// TIA Portal V19 export
FUNCTION_BLOCK "A0302_Spintore_FB"   // FB91, LAD
// stored: MemoryReserve 100, SetENOAutomatically false
   VAR_INPUT
      AreaInterface : "AreaInterface";
      ZSI : "udt_ZoneSafetyInterface";
      DSI_Feed : "udt_DeviceSafetyInterface";
      DSI_Valve : "udt_DeviceSafetyInterface";
      Drive : "TAx_DriveInterface";
      DataIn : Struct
         OP : "OP_PB";
         P5 { ExternalAccessible := 'False'; ExternalVisible := 'False'; ExternalWritable := 'False'} : Struct
            Orz_AnalSens : Int;
            FTC_FuoriIngombro_A0301 : Bool;   // FTC fuori ingombro lato bordatrice
         END_STRUCT;
      END_STRUCT;
      Cin : Struct
         Manager { ExternalWritable := 'False'} : Struct
            EnableStopDoorOpeningReq : Bool;
            EnableStopInPhase : Bool;
            EnableStopProgrammed : Bool;
            Control_ON : Bool;
            REST_Req : Bool;
            WORK_Req : Bool;
            Rest : Bool;
            Work : Bool;
         END_STRUCT;
         SemiAut_Pb { ExternalAccessible := 'False'; ExternalVisible := 'False'; ExternalWritable := 'False'} : Bool;
         P4 { ExternalWritable := 'False'} : Struct
            Fermi : "ValveMachine_COut";
         END_STRUCT;
         P5 { ExternalWritable := 'False'} : Struct
            "En/Dis_SpinLat_2" : Bool;   // 1=Enable / 0=Disable
            QuotaIngombro_SpinLat2 : Real;
            QuotaIngombro_SpinLat1 : Real;
            Spintore_Lat : Struct
               Spin_Lat1 : Struct
                  Standstill : Bool;
                  Rest_CheckNext : Bool;
                  Work_CheckNext : Bool;
                  Rest : Bool;
                  Work : Bool;
               END_STRUCT;
               Spin_Lat2 : Struct
                  Standstill : Bool;
                  Rest_CheckNext : Bool;
                  Work_CheckNext : Bool;
                  Rest : Bool;
                  Work : Bool;
               END_STRUCT;
               Vrt_1 : "ValveMachine_COut";
               Orz_1 : "ValveMachine_COut";
               Vrt_2 : "ValveMachine_COut";
               Orz_2 : "ValveMachine_COut";
               Sollevatori : "ValveMachine_COut";
            END_STRUCT;
         END_STRUCT;
         Trasporto { ExternalAccessible := 'False'; ExternalVisible := 'False'; ExternalWritable := 'False'} : "SpeedMachine_COut";
         Bordatrice : Struct   // *************************
            Ax : "Positioning_EPOS_Machine_COut";
            TargetVel : LReal;
            Perc_Vel : LReal;
            Sens : Struct
               FTC_Uscita : Bool;
            END_STRUCT;
         END_STRUCT;
      END_STRUCT;
      Config : Struct
         Ax : "Positioning_EPOS_Machine_Config_NEW";
         Vrt : "ValveMachine_Config";
         Orz : "ValveMachine_Config";
         SpintoreLat : Struct
            QuotaIngombro_SpinLat2 : Real := 2705.0;
            QuotaIngombro_SpinLat1 : Real := 4777.0;
         END_STRUCT;
         Bordatrice : Struct
            QuotaIngresso : Real := 600.0;
         END_STRUCT;
         DelayMissingCondition : Time;
      END_STRUCT;
      HWID_Ax_TEL111 : HW_SUBMODULE;
   END_VAR
   VAR_OUTPUT
      MachineInterface : "MachineInterface";
      DataOut : "Positioning_EPOS_Machine_DataOut";
      COut : Struct
         Ax_Sts : Struct
            PosAttesa_Reached : Bool;
            PosFineSpinta_Reached : Bool;
         END_STRUCT;
         Ax : "Positioning_EPOS_Machine_COut";
         Spintore : "ValveMachine_COut";
         Vrt : "ValveMachine_COut";
         Orz : "ValveMachine_COut";
      END_STRUCT;
   END_VAR
   VAR_IN_OUT
      Par : Struct
         Sens : "Analogic_SensorManagement_Par";
      END_STRUCT;
      Data : Struct
         Sens : "Analogic_SensorManagement_Data";
         HMI : "HMI_Preset";
         Ax_Pos : "A0301_Mach_Ax_Pos_Data";
      END_STRUCT;
      Par_Mach : "A0301_Mach_Sens_Par";
      Par_Ax_Manu : "Positioning_EPOS_Machine_Par";
      Pers_Data : Struct
         EncoderAbsolute_Preset_OK : Bool;
         Persistent_ActualPosition : LReal;
      END_STRUCT;
      Par_Ax_Auto : "A0301_Mach_Speed_Par";
   END_VAR
   VAR
      Alarm : Struct
         Ax : "Positioning_EPOS_Machine_Alr";
         Ax_NeedPreset { S7_SetPoint := 'True'} : Bool;
         Vrt : "ValveAlr";
         Orz : "ValveAlr";
         Orz_AnalSens_Issue : Bool;
         Orz_AnalSens_Compressed : Bool;
      END_STRUCT;
      Warning : Struct
         Ax : "Positioning_EPOS_Machine_Wng";
         Vrt : "ValveMachine_Wng";
         Orz { S7_SetPoint := 'True'} : "ValveMachine_Wng";
         Orz_AnalSens { S7_SetPoint := 'True'} : "Analogic_SensorManagement_Warning";
         OP_REST_MissingCnd : Bool;   // Mancanza comando arresto
         OP_WORK_MissingCnd : Bool;   // Mancanza consenso lavoro
      END_STRUCT;
      Sts : Struct
         ReadyForMove : Bool;   // Pronto al movimento
         OP_CanMoveFreely : Bool;
         OP_Ax_Rest_Cnd : Bool;
         OP_Ax_Work_Cnd : Bool;
         OP_Spin_Rest_Cnd : Bool;
         OP_Spin_Work_Cnd : Bool;
         A0301_Beam_BLean : Real;
         A0302_Beam_BLean : Real;
         Vrt_Work_ExtEnable : Bool;
         Orz_Work_ExtEnable : Bool;
      END_STRUCT;
      Ctrl : Struct
         SpinVrtOrz : Struct
            OP_Rest_Man : Bool;
            OP_Work_Man : Bool;
            OP_Rest_Aut : Bool;
            OP_Work_Aut : Bool;
            OP_Rest : Bool;
            OP_Work : Bool;
         END_STRUCT;
         Ax : Struct
            OP_Rest_Man : Bool;
            OP_Work_Man : Bool;
            OP_Rest_Aut : Bool;
            OP_Work_Aut : Bool;
            OP_Rest : Bool;
            OP_Work : Bool;
            Vel : LReal;
            VelMax : Real;
            Dec : LReal;
         END_STRUCT;
      END_STRUCT;
      HMI : Struct
         Ax : "AnalogSens_HmiData";
         Orz_AnalSens_PB_Preset { ExternalAccessible := 'False'; ExternalVisible := 'False'; ExternalWritable := 'False'} : Bool;   // Pulsante Preset value
         Orz_AnalSens_Preset_Value : LReal;
      END_STRUCT;
      Ax { S7_SetPoint := 'True'} : "Positioning_EPOS_Machine_FB_NEW";   // Spintore longitudinale
      Vrt { S7_SetPoint := 'True'} : "ValveMachine_FB";   // Sollevatore verticale
      Orz { S7_SetPoint := 'True'} : "ValveMachine_FB";   // Compensatore orizzontale
      Orz_AnalSens { S7_SetPoint := 'True'} : "Analogic_SensorManagement";
      ValueBLeanOvr : Array[1..15] of Real;
      IEC : Struct
         TON_DelayFTC_Ingombro_A0301 : IEC_TIMER;
         TOF_DelayFTC_Ingombro_A0301 { S7_SetPoint := 'True'} : IEC_TIMER;
         FTC_On { S7_SetPoint := 'True'} : Bool;
      END_STRUCT;
      AUX : Struct
         OP_Rest_PB : Bool;
         OP_Work_PB : Bool;
      END_STRUCT;
      TON_OP_REST_MissingCnd { S7_SetPoint := 'True'} : TON_TIME;
      TON_OP_WORK_MissingCnd { S7_SetPoint := 'True'} : TON_TIME;
      BTrk_Item : Struct
         BLean : Real;
         O_ID : DInt;
      END_STRUCT;
   END_VAR
   VAR_TEMP
      i : Int;
      DecMax : LReal;
      Orz_SpazioSafe : LReal;
      Calcoli : Struct
         SUB_SpinLat2 : LReal;
         SUB_SpinLat1 : LReal;
         Pos_Target_2 : LReal;
         Pos_Target_1 : LReal;
         Ax_Target : LReal;
      END_STRUCT;
      PE : Struct
         OP_Rest_PB : Bool;
         OP_Work_PB : Bool;
      END_STRUCT;
      BTrk_GetData_A0302 : Struct
         indx : Int;   // Se trovato tra i TODO / ENDING / OUT questo è l'indice dove sono stati prelevati i dati
         Sts : Int;   // 0 = Non Trovato; 0 = ACT; 1 = TODO; 2=ENDING; 3 = OUT
         Item : "Prod_Item_small";
      END_STRUCT;
      BTrk_GetData_A0301 : Struct
         indx : Int;   // Se trovato tra i TODO / ENDING / OUT questo è l'indice dove sono stati prelevati i dati
         Sts : Int;   // 0 = Non Trovato; 0 = ACT; 1 = TODO; 2=ENDING; 3 = OUT
         Item : "Prod_Item_small";
      END_STRUCT;
      Stop_Ax_SpinLong : Bool;
      GetData_A0301_B : Bool;
      GetData_A0302_In : Bool;
   END_VAR
   VAR CONSTANT
      Offset_SpinLong_To_SpinLat2 : Real;   // Offset calcolato da quota ingombro Spintore Laterale2 per bloccare Spintore Longitudinale e allarme se SpinLat2 alto
      Offset_SpinLong_To_SpinLat1 : Real;   // Offset calcolato da quota ingombro Spintore Laterale1 per bloccare Spintore Longitudinale e allarme se SpinLat1 alto
   END_VAR
   // Orz_AnalSens.Filter.Tau := T#10ms;
   VAR_TEMP   // added for the SCL form of the ladder/FBD networks
      _w1 : Bool;
      _w2 : Bool;
      _w3 : Bool;
      _w4 : Bool;
      _w5 : Bool;
      _w6 : Bool;
   END_VAR
BEGIN

REGION Network 1 (SCL): Reset allarmi
   IF #AreaInterface.RstAlarms THEN
       #Alarm.Orz_AnalSens_Issue := FALSE;
       #Warning.Orz_AnalSens.SignalError := FALSE;
   END_IF;
END_REGION

REGION Network 2: <+>
END_REGION

REGION Network 4: CONTROLLO MES lunghezza Beams
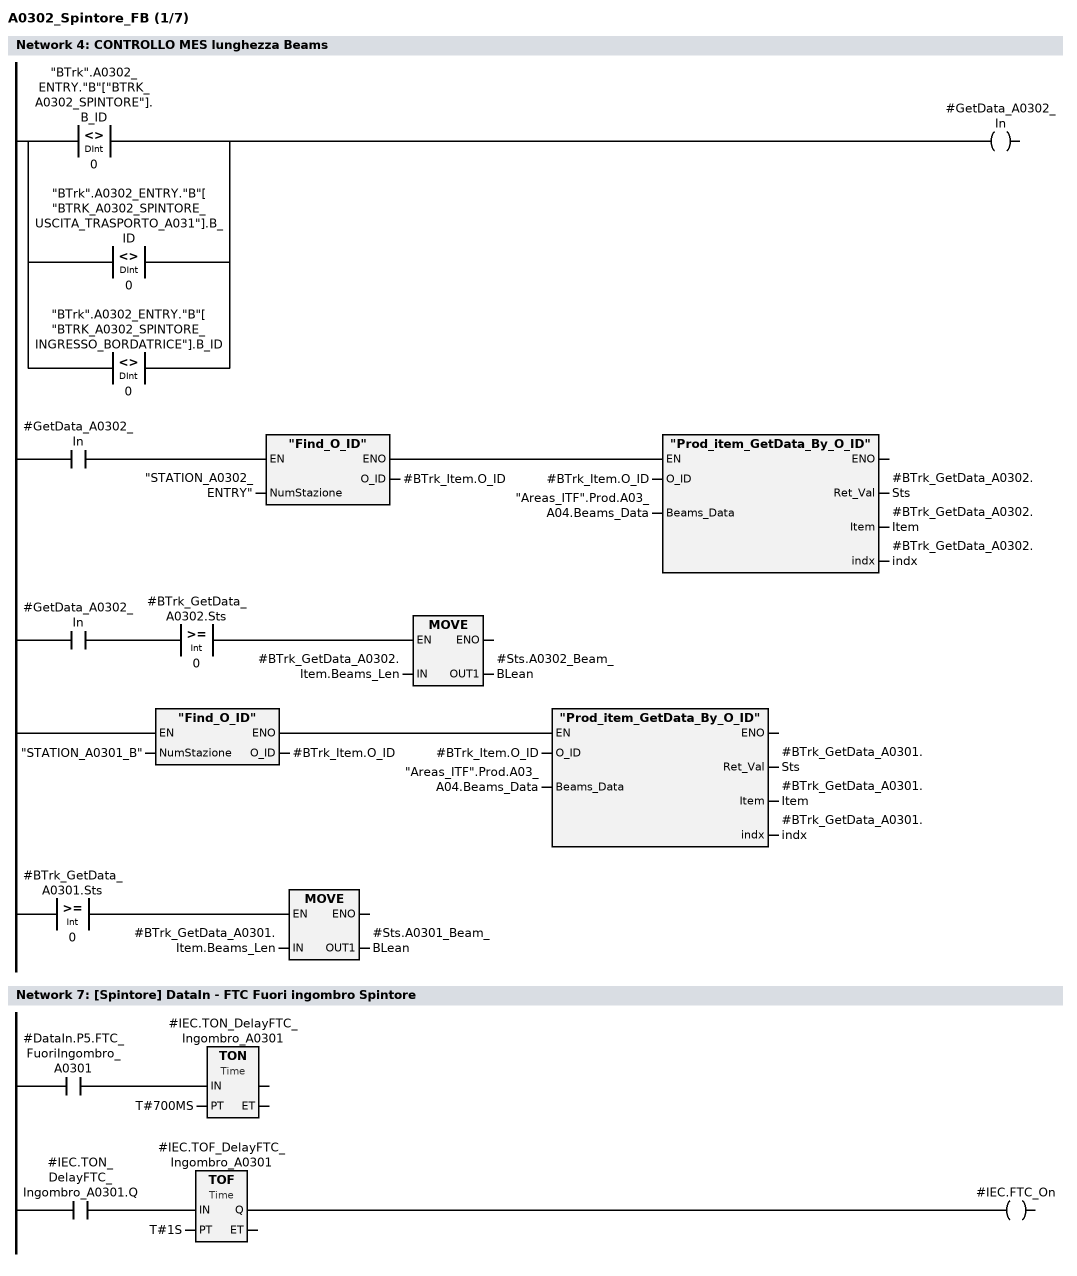
   RUNG wire#powerrail
      { S7_Templates := "SrcType := DInt" } NE_Contact(in1 := "BTrk".A0302_ENTRY."B"["BTRK_A0302_SPINTORE"].B_ID, in2 := 0)
      wire#w1
      Coil( #GetData_A0302_In )
   END_RUNG
   RUNG wire#powerrail
      { S7_Templates := "SrcType := DInt" } NE_Contact(in1 := "BTrk".A0302_ENTRY."B"["BTRK_A0302_SPINTORE_USCITA_TRASPORTO_A031"].B_ID, in2 := 0)
   END_RUNG wire#w1
   RUNG wire#powerrail
      { S7_Templates := "SrcType := DInt" } NE_Contact(in1 := "BTrk".A0302_ENTRY."B"["BTRK_A0302_SPINTORE_INGRESSO_BORDATRICE"].B_ID, in2 := 0)
   END_RUNG wire#w1
   RUNG wire#powerrail
      Contact( #GetData_A0302_In )
      "Find_O_ID"(NumStazione := "STATION_A0302_ENTRY", O_ID => #BTrk_Item.O_ID)
      "Prod_item_GetData_By_O_ID"(O_ID := #BTrk_Item.O_ID, Beams_Data := "Areas_ITF".Prod.A03_A04.Beams_Data, Ret_Val => #BTrk_GetData_A0302.Sts, Item => #BTrk_GetData_A0302.Item, indx => #BTrk_GetData_A0302.indx)
   END_RUNG
   RUNG wire#powerrail
      Contact( #GetData_A0302_In )
      { S7_Templates := "SrcType := Int" } GE_Contact(in1 := #BTrk_GetData_A0302.Sts, in2 := 0)
      Move(in := #BTrk_GetData_A0302.Item.Beams_Len, out1 => #Sts.A0302_Beam_BLean)
   END_RUNG
   RUNG wire#powerrail
      "Find_O_ID"(NumStazione := "STATION_A0301_B", O_ID => #BTrk_Item.O_ID)
      "Prod_item_GetData_By_O_ID"(O_ID := #BTrk_Item.O_ID, Beams_Data := "Areas_ITF".Prod.A03_A04.Beams_Data, Ret_Val => #BTrk_GetData_A0301.Sts, Item => #BTrk_GetData_A0301.Item, indx => #BTrk_GetData_A0301.indx)
   END_RUNG
   RUNG wire#powerrail
      { S7_Templates := "SrcType := Int" } GE_Contact(in1 := #BTrk_GetData_A0301.Sts, in2 := 0)
      Move(in := #BTrk_GetData_A0301.Item.Beams_Len, out1 => #Sts.A0301_Beam_BLean)
   END_RUNG
   // the same network as SCL:
   #GetData_A0302_In := ("BTrk".A0302_ENTRY."B"["BTRK_A0302_SPINTORE"].B_ID <> 0) OR ("BTrk".A0302_ENTRY."B"["BTRK_A0302_SPINTORE_USCITA_TRASPORTO_A031"].B_ID <> 0) OR ("BTrk".A0302_ENTRY."B"["BTRK_A0302_SPINTORE_INGRESSO_BORDATRICE"].B_ID <> 0);
   "Find_O_ID"(EN := #GetData_A0302_In,
               NumStazione := "STATION_A0302_ENTRY",
               O_ID => #BTrk_Item.O_ID,
               ENO => #_w1);
   IF #_w1 THEN
       #BTrk_GetData_A0302.Sts := "Prod_item_GetData_By_O_ID"(O_ID := #BTrk_Item.O_ID,
                               Beams_Data := "Areas_ITF".Prod.A03_A04.Beams_Data,
                               Item => #BTrk_GetData_A0302.Item,
                               indx => #BTrk_GetData_A0302.indx);
   END_IF;
   IF #GetData_A0302_In AND (#BTrk_GetData_A0302.Sts >= 0) THEN
       #Sts.A0302_Beam_BLean := #BTrk_GetData_A0302.Item.Beams_Len;
   END_IF;
   "Find_O_ID"(NumStazione := "STATION_A0301_B", O_ID => #BTrk_Item.O_ID, ENO => #_w2);
   IF #_w2 THEN
       #BTrk_GetData_A0301.Sts := "Prod_item_GetData_By_O_ID"(O_ID := #BTrk_Item.O_ID,
                               Beams_Data := "Areas_ITF".Prod.A03_A04.Beams_Data,
                               Item => #BTrk_GetData_A0301.Item,
                               indx => #BTrk_GetData_A0301.indx);
   END_IF;
   IF #BTrk_GetData_A0301.Sts >= 0 THEN #Sts.A0301_Beam_BLean := #BTrk_GetData_A0301.Item.Beams_Len; END_IF;
END_REGION

REGION Network 5 (SCL): CALCOLI - Posizioni Attesa / Spinta per lavoro Spintore

   #BTrk_GetData_A0302.Item.O_ID := #BTrk_GetData_A0302.Item.O_ID;
   #BTrk_Item.BLean:=#BTrk_GetData_A0302.Item.Beams_Len;
   // ***********************************************************************************************************
   // 
   REGION POSIZIONE ATTESA PEZZO IN ENTRATA

       // Se ho una misura traking vado in posizionamento calcolando la misura del Beams più alta + Offset sennò vado indietro fino a pos. minima
       IF #Sts.A0301_Beam_BLean <> 0 THEN
           #Data.Ax_Pos.PosAttesa := (#Ax.COut.MaxPosition -#Sts.A0301_Beam_BLean) - (#Data.Ax_Pos.OffsetPosAttesa - #Config.Bordatrice.QuotaIngresso);
       ELSIF #Sts.OP_CanMoveFreely THEN
           #BTrk_Item.BLean := 0;
           #Data.Ax_Pos.PosAttesa := ( #Ax.COut.MinPosition) + #Data.Ax_Pos.OffsetPosAttesa;
       END_IF;

   END_REGION ;
   //
   // ***********************************************************************************************************
   // 
   REGION POSIZIONE FINE SPINTA PEZZO IN USCITA

       // CALCOLO Pos.Fine Spinta Target finale
       IF #Sts.A0302_Beam_BLean <> 0 THEN
           #Data.Ax_Pos.PosFineSpinta := (#Ax.COut.MaxPosition - #Sts.A0302_Beam_BLean) + (#Config.Bordatrice.QuotaIngresso);
       ELSIF #BTrk_Item.BLean = 0 THEN
           #Data.Ax_Pos.PosFineSpinta := (#Ax.COut.MaxPosition - #Data.Ax_Pos.OffsetPosAttesa);
       END_IF;

       (*
       // CALCOLO differenza tra Pos.Attesa e Quota ingombro Spintore laterale 2 SE incluso 
       IF #Cin.P5."En/Dis_SpinLat_2"
           AND #Ax.COut.ActualPosition < (#Config.SpintoreLat.QuotaIngombro_SpinLat2 +  #Config.SpintoreLat.OffsetPosAttesa) THEN
           #Calcoli.SUB_SpinLat2 :=((#Data.Ax_Pos.PosAttesa) + (#Config.SpintoreLat.QuotaIngombro_SpinLat2));
       END_IF;

       // CALCOLO differenza tra Pos.Attesa e Quota ingombro Spintore laterale 1 
       IF #Ax.COut.ActualPosition > #Config.SpintoreLat.QuotaIngombro_SpinLat1 THEN
           #Calcoli.SUB_SpinLat1 :=((#Data.Ax_Pos.PosAttesa) + (#Config.SpintoreLat.QuotaIngombro_SpinLat1));
       END_IF;

       // CALCOLI Posizioni Target SPINTORI LATERALI
       #Calcoli.Pos_Target_2 := (#Data.Ax_Pos.PosAttesa) + (#Calcoli.SUB_SpinLat2);
       #Calcoli.Pos_Target_1 := (#Data.Ax_Pos.PosAttesa) + (#Calcoli.SUB_SpinLat1);

       // SPINTORE LATERALE 1&2 - AX - POS. Target
       IF #Cin.P5."En/Dis_SpinLat_2"
           AND #Data.Ax_Pos.PosFineSpinta >= #Calcoli.Pos_Target_2 THEN
           #Calcoli.Ax_Target := #Calcoli.Pos_Target_2;
       ELSIF #Data.Ax_Pos.PosFineSpinta >= #Calcoli.Pos_Target_1
           AND #Ax.COut.ActualPosition < (-#Config.SpintoreLat.QuotaIngombro_SpinLat2) THEN
           #Calcoli.Ax_Target := #Calcoli.Pos_Target_1;
       ELSIF #Ax.#COut.ActualPosition < (-#Config.SpintoreLat.QuotaIngombro_SpinLat1) THEN
           #Calcoli.Ax_Target := #Data.Ax_Pos.PosFineSpinta;
       END_IF;
       *)

   END_REGION ;
   //
   // ***********************************************************************************************************
END_REGION

REGION Network 6: <+>
END_REGION

REGION Network 7: [Spintore] DataIn - FTC Fuori ingombro Spintore
   RUNG wire#powerrail
      Contact( #DataIn.P5.FTC_FuoriIngombro_A0301 )
      { S7_Templates := "time_type := Time" } #IEC.TON_DelayFTC_Ingombro_A0301.TON(pt := T#700MS, et =>)
   END_RUNG
   RUNG wire#powerrail
      Contact( #IEC.TON_DelayFTC_Ingombro_A0301.Q )
      { S7_Templates := "time_type := Time" } #IEC.TOF_DelayFTC_Ingombro_A0301.TOF(pt := T#1S, et =>)
      Coil( #IEC.FTC_On )
   END_RUNG
   // the same network as SCL:
   #IEC.TON_DelayFTC_Ingombro_A0301.TON(IN := #DataIn.P5.FTC_FuoriIngombro_A0301, PT := T#700MS);
   #IEC.TOF_DelayFTC_Ingombro_A0301.TOF(IN := #IEC.TON_DelayFTC_Ingombro_A0301.Q, PT := T#1S);
   #IEC.FTC_On := #IEC.TOF_DelayFTC_Ingombro_A0301.Q;
END_REGION

REGION Network 8: <+>
END_REGION

REGION Network 9: Operazione può muoversi liberamente perchè non sposta nessun BEAM
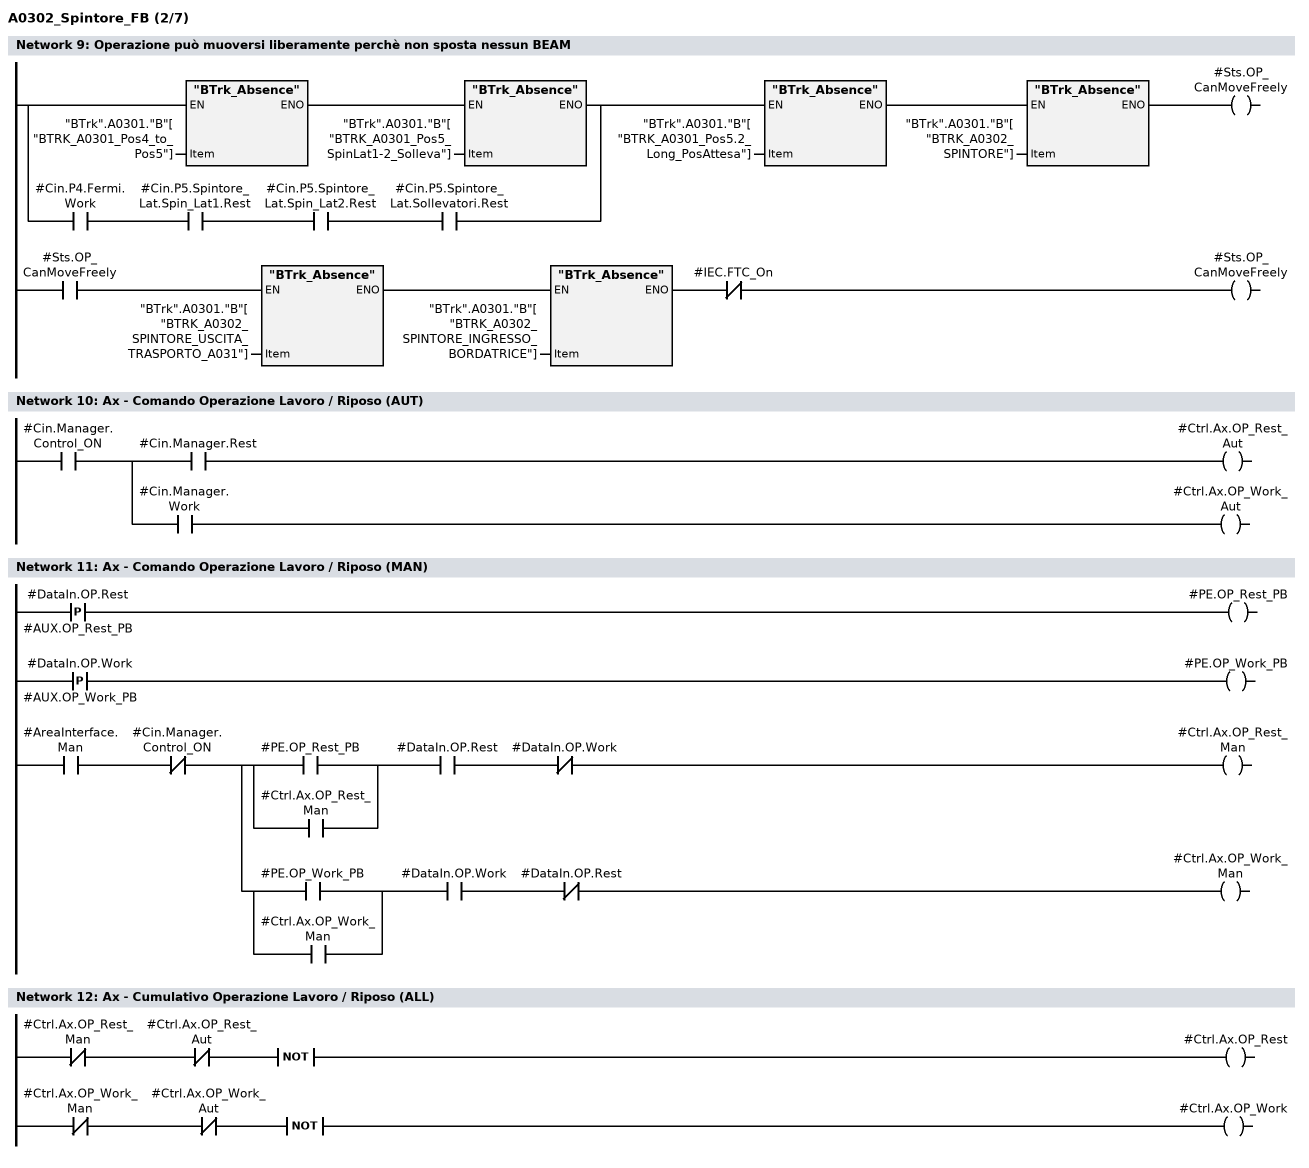
   RUNG wire#powerrail
      "BTrk_Absence"(Item := "BTrk".A0301."B"["BTRK_A0301_Pos4_to_Pos5"])
      "BTrk_Absence"(Item := "BTrk".A0301."B"["BTRK_A0301_Pos5_SpinLat1-2_Solleva"])
      wire#w1
      "BTrk_Absence"(Item := "BTrk".A0301."B"["BTRK_A0301_Pos5.2_Long_PosAttesa"])
      "BTrk_Absence"(Item := "BTrk".A0301."B"["BTRK_A0302_SPINTORE"])
      Coil( #Sts.OP_CanMoveFreely )
   END_RUNG
   RUNG wire#powerrail
      Contact( #Cin.P4.Fermi.Work )
      Contact( #Cin.P5.Spintore_Lat.Spin_Lat1.Rest )
      Contact( #Cin.P5.Spintore_Lat.Spin_Lat2.Rest )
      Contact( #Cin.P5.Spintore_Lat.Sollevatori.Rest )
   END_RUNG wire#w1
   RUNG wire#powerrail
      Contact( #Sts.OP_CanMoveFreely )
      "BTrk_Absence"(Item := "BTrk".A0301."B"["BTRK_A0302_SPINTORE_USCITA_TRASPORTO_A031"])
      "BTrk_Absence"(Item := "BTrk".A0301."B"["BTRK_A0302_SPINTORE_INGRESSO_BORDATRICE"])
      I_Contact( #IEC.FTC_On )
      Coil( #Sts.OP_CanMoveFreely )
   END_RUNG
   // the same network as SCL:
   "BTrk_Absence"(Item := "BTrk".A0301."B"["BTRK_A0301_Pos4_to_Pos5"], ENO => #_w1);
   "BTrk_Absence"(EN := #_w1, Item := "BTrk".A0301."B"["BTRK_A0301_Pos5_SpinLat1-2_Solleva"], ENO => #_w2);
   "BTrk_Absence"(EN := #_w2 OR (#Cin.P4.Fermi.Work AND #Cin.P5.Spintore_Lat.Spin_Lat1.Rest AND #Cin.P5.Spintore_Lat.Spin_Lat2.Rest AND #Cin.P5.Spintore_Lat.Sollevatori.Rest),
                  Item := "BTrk".A0301."B"["BTRK_A0301_Pos5.2_Long_PosAttesa"],
                  ENO => #_w3);
   "BTrk_Absence"(EN := #_w3, Item := "BTrk".A0301."B"["BTRK_A0302_SPINTORE"], ENO => #_w4);
   #Sts.OP_CanMoveFreely := #_w4;
   "BTrk_Absence"(EN := #Sts.OP_CanMoveFreely,
                  Item := "BTrk".A0301."B"["BTRK_A0302_SPINTORE_USCITA_TRASPORTO_A031"],
                  ENO => #_w5);
   "BTrk_Absence"(EN := #_w5, Item := "BTrk".A0301."B"["BTRK_A0302_SPINTORE_INGRESSO_BORDATRICE"], ENO => #_w6);
   #Sts.OP_CanMoveFreely := #_w6 AND NOT #IEC.FTC_On;
END_REGION

REGION Network 10: Ax - Comando Operazione Lavoro / Riposo (AUT)
   RUNG wire#powerrail
      Contact( #Cin.Manager.Control_ON )
      wire#w1
      Contact( #Cin.Manager.Rest )
      Coil( #Ctrl.Ax.OP_Rest_Aut )
   END_RUNG
   RUNG wire#w1
      Contact( #Cin.Manager.Work )
      Coil( #Ctrl.Ax.OP_Work_Aut )
   END_RUNG
   // the same network as SCL:
   #Ctrl.Ax.OP_Rest_Aut := #Cin.Manager.Control_ON AND #Cin.Manager.Rest;
   #Ctrl.Ax.OP_Work_Aut := #Cin.Manager.Control_ON AND #Cin.Manager.Work;
END_REGION

REGION Network 11: Ax - Comando Operazione Lavoro / Riposo (MAN)
   RUNG wire#powerrail
      P_Contact(operand := #DataIn.OP.Rest, bit := #AUX.OP_Rest_PB)
      Coil( #PE.OP_Rest_PB )
   END_RUNG
   RUNG wire#powerrail
      P_Contact(operand := #DataIn.OP.Work, bit := #AUX.OP_Work_PB)
      Coil( #PE.OP_Work_PB )
   END_RUNG
   RUNG wire#powerrail
      Contact( #AreaInterface.Man )
      I_Contact( #Cin.Manager.Control_ON )
      wire#w1
      Contact( #PE.OP_Rest_PB )
      wire#w2
      Contact( #DataIn.OP.Rest )
      I_Contact( #DataIn.OP.Work )
      Coil( #Ctrl.Ax.OP_Rest_Man )
   END_RUNG
   RUNG wire#w1
      Contact( #Ctrl.Ax.OP_Rest_Man )
   END_RUNG wire#w2
   RUNG wire#w1
      Contact( #PE.OP_Work_PB )
      wire#w3
      Contact( #DataIn.OP.Work )
      I_Contact( #DataIn.OP.Rest )
      Coil( #Ctrl.Ax.OP_Work_Man )
   END_RUNG
   RUNG wire#w1
      Contact( #Ctrl.Ax.OP_Work_Man )
   END_RUNG wire#w3
   // the same network as SCL:
   #_w1 := #DataIn.OP.Rest AND NOT #AUX.OP_Rest_PB;   // rising edge of #DataIn.OP.Rest
   #AUX.OP_Rest_PB := #DataIn.OP.Rest;
   #PE.OP_Rest_PB := #_w1;
   #_w2 := #DataIn.OP.Work AND NOT #AUX.OP_Work_PB;   // rising edge of #DataIn.OP.Work
   #AUX.OP_Work_PB := #DataIn.OP.Work;
   #PE.OP_Work_PB := #_w2;
   #_w3 := #AreaInterface.Man AND NOT #Cin.Manager.Control_ON;
   #Ctrl.Ax.OP_Rest_Man := #_w3 AND (#PE.OP_Rest_PB OR #Ctrl.Ax.OP_Rest_Man) AND #DataIn.OP.Rest AND NOT #DataIn.OP.Work;
   #Ctrl.Ax.OP_Work_Man := #_w3 AND (#PE.OP_Work_PB OR #Ctrl.Ax.OP_Work_Man) AND #DataIn.OP.Work AND NOT #DataIn.OP.Rest;
END_REGION

REGION Network 12: Ax - Cumulativo Operazione Lavoro / Riposo (ALL)
   RUNG wire#powerrail
      I_Contact( #Ctrl.Ax.OP_Rest_Man )
      I_Contact( #Ctrl.Ax.OP_Rest_Aut )
      Not()
      Coil( #Ctrl.Ax.OP_Rest )
   END_RUNG
   RUNG wire#powerrail
      I_Contact( #Ctrl.Ax.OP_Work_Man )
      I_Contact( #Ctrl.Ax.OP_Work_Aut )
      Not()
      Coil( #Ctrl.Ax.OP_Work )
   END_RUNG
   // the same network as SCL:
   #Ctrl.Ax.OP_Rest := NOT (NOT #Ctrl.Ax.OP_Rest_Man AND NOT #Ctrl.Ax.OP_Rest_Aut);
   #Ctrl.Ax.OP_Work := NOT (NOT #Ctrl.Ax.OP_Work_Man AND NOT #Ctrl.Ax.OP_Work_Aut);
END_REGION

REGION Network 13: Ax - Condizioni movimento Operazione a Lavoro / Riposo
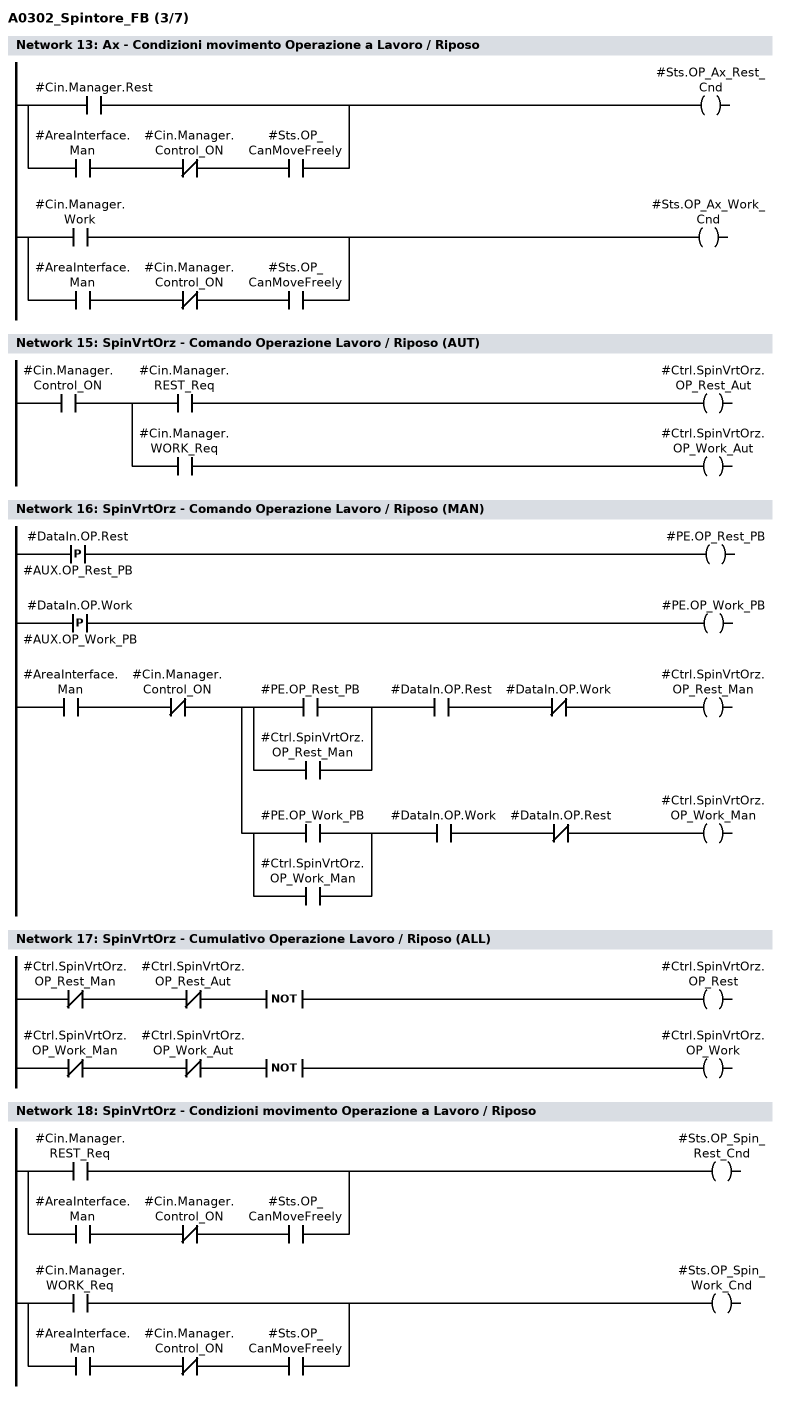
   RUNG wire#powerrail
      Contact( #Cin.Manager.Rest )
      wire#w1
      Coil( #Sts.OP_Ax_Rest_Cnd )
   END_RUNG
   RUNG wire#powerrail
      Contact( #AreaInterface.Man )
      I_Contact( #Cin.Manager.Control_ON )
      Contact( #Sts.OP_CanMoveFreely )
   END_RUNG wire#w1
   RUNG wire#powerrail
      Contact( #Cin.Manager.Work )
      wire#w2
      Coil( #Sts.OP_Ax_Work_Cnd )
   END_RUNG
   RUNG wire#powerrail
      Contact( #AreaInterface.Man )
      I_Contact( #Cin.Manager.Control_ON )
      Contact( #Sts.OP_CanMoveFreely )
   END_RUNG wire#w2
   // the same network as SCL:
   #Sts.OP_Ax_Rest_Cnd := #Cin.Manager.Rest OR (#AreaInterface.Man AND NOT #Cin.Manager.Control_ON AND #Sts.OP_CanMoveFreely);
   #Sts.OP_Ax_Work_Cnd := #Cin.Manager.Work OR (#AreaInterface.Man AND NOT #Cin.Manager.Control_ON AND #Sts.OP_CanMoveFreely);
END_REGION

REGION Network 15: SpinVrtOrz - Comando Operazione Lavoro / Riposo (AUT)
   RUNG wire#powerrail
      Contact( #Cin.Manager.Control_ON )
      wire#w1
      Contact( #Cin.Manager.REST_Req )
      Coil( #Ctrl.SpinVrtOrz.OP_Rest_Aut )
   END_RUNG
   RUNG wire#w1
      Contact( #Cin.Manager.WORK_Req )
      Coil( #Ctrl.SpinVrtOrz.OP_Work_Aut )
   END_RUNG
   // the same network as SCL:
   #Ctrl.SpinVrtOrz.OP_Rest_Aut := #Cin.Manager.Control_ON AND #Cin.Manager.REST_Req;
   #Ctrl.SpinVrtOrz.OP_Work_Aut := #Cin.Manager.Control_ON AND #Cin.Manager.WORK_Req;
END_REGION

REGION Network 16: SpinVrtOrz - Comando Operazione Lavoro / Riposo (MAN)
   RUNG wire#powerrail
      P_Contact(operand := #DataIn.OP.Rest, bit := #AUX.OP_Rest_PB)
      Coil( #PE.OP_Rest_PB )
   END_RUNG
   RUNG wire#powerrail
      P_Contact(operand := #DataIn.OP.Work, bit := #AUX.OP_Work_PB)
      Coil( #PE.OP_Work_PB )
   END_RUNG
   RUNG wire#powerrail
      Contact( #AreaInterface.Man )
      I_Contact( #Cin.Manager.Control_ON )
      wire#w1
      Contact( #PE.OP_Rest_PB )
      wire#w2
      Contact( #DataIn.OP.Rest )
      I_Contact( #DataIn.OP.Work )
      Coil( #Ctrl.SpinVrtOrz.OP_Rest_Man )
   END_RUNG
   RUNG wire#w1
      Contact( #Ctrl.SpinVrtOrz.OP_Rest_Man )
   END_RUNG wire#w2
   RUNG wire#w1
      Contact( #PE.OP_Work_PB )
      wire#w3
      Contact( #DataIn.OP.Work )
      I_Contact( #DataIn.OP.Rest )
      Coil( #Ctrl.SpinVrtOrz.OP_Work_Man )
   END_RUNG
   RUNG wire#w1
      Contact( #Ctrl.SpinVrtOrz.OP_Work_Man )
   END_RUNG wire#w3
   // the same network as SCL:
   #_w1 := #DataIn.OP.Rest AND NOT #AUX.OP_Rest_PB;   // rising edge of #DataIn.OP.Rest
   #AUX.OP_Rest_PB := #DataIn.OP.Rest;
   #PE.OP_Rest_PB := #_w1;
   #_w2 := #DataIn.OP.Work AND NOT #AUX.OP_Work_PB;   // rising edge of #DataIn.OP.Work
   #AUX.OP_Work_PB := #DataIn.OP.Work;
   #PE.OP_Work_PB := #_w2;
   #_w3 := #AreaInterface.Man AND NOT #Cin.Manager.Control_ON;
   #Ctrl.SpinVrtOrz.OP_Rest_Man := #_w3 AND (#PE.OP_Rest_PB OR #Ctrl.SpinVrtOrz.OP_Rest_Man) AND #DataIn.OP.Rest AND NOT #DataIn.OP.Work;
   #Ctrl.SpinVrtOrz.OP_Work_Man := #_w3 AND (#PE.OP_Work_PB OR #Ctrl.SpinVrtOrz.OP_Work_Man) AND #DataIn.OP.Work AND NOT #DataIn.OP.Rest;
END_REGION

REGION Network 17: SpinVrtOrz - Cumulativo Operazione Lavoro / Riposo (ALL)
   RUNG wire#powerrail
      I_Contact( #Ctrl.SpinVrtOrz.OP_Rest_Man )
      I_Contact( #Ctrl.SpinVrtOrz.OP_Rest_Aut )
      Not()
      Coil( #Ctrl.SpinVrtOrz.OP_Rest )
   END_RUNG
   RUNG wire#powerrail
      I_Contact( #Ctrl.SpinVrtOrz.OP_Work_Man )
      I_Contact( #Ctrl.SpinVrtOrz.OP_Work_Aut )
      Not()
      Coil( #Ctrl.SpinVrtOrz.OP_Work )
   END_RUNG
   // the same network as SCL:
   #Ctrl.SpinVrtOrz.OP_Rest := NOT (NOT #Ctrl.SpinVrtOrz.OP_Rest_Man AND NOT #Ctrl.SpinVrtOrz.OP_Rest_Aut);
   #Ctrl.SpinVrtOrz.OP_Work := NOT (NOT #Ctrl.SpinVrtOrz.OP_Work_Man AND NOT #Ctrl.SpinVrtOrz.OP_Work_Aut);
END_REGION

REGION Network 18: SpinVrtOrz - Condizioni movimento Operazione a Lavoro / Riposo
   RUNG wire#powerrail
      Contact( #Cin.Manager.REST_Req )
      wire#w1
      Coil( #Sts.OP_Spin_Rest_Cnd )
   END_RUNG
   RUNG wire#powerrail
      Contact( #AreaInterface.Man )
      I_Contact( #Cin.Manager.Control_ON )
      Contact( #Sts.OP_CanMoveFreely )
   END_RUNG wire#w1
   RUNG wire#powerrail
      Contact( #Cin.Manager.WORK_Req )
      wire#w2
      Coil( #Sts.OP_Spin_Work_Cnd )
   END_RUNG
   RUNG wire#powerrail
      Contact( #AreaInterface.Man )
      I_Contact( #Cin.Manager.Control_ON )
      Contact( #Sts.OP_CanMoveFreely )
   END_RUNG wire#w2
   // the same network as SCL:
   #Sts.OP_Spin_Rest_Cnd := #Cin.Manager.REST_Req OR (#AreaInterface.Man AND NOT #Cin.Manager.Control_ON AND #Sts.OP_CanMoveFreely);
   #Sts.OP_Spin_Work_Cnd := #Cin.Manager.WORK_Req OR (#AreaInterface.Man AND NOT #Cin.Manager.Control_ON AND #Sts.OP_CanMoveFreely);
END_REGION

REGION Network 20 (SCL): Verticale + Orizzontale + Ax - Cin Manager (Esecuzione sequenza comandi)
   #Ax.CIn.Manager.Control_ON:= #Cin.Manager.Control_ON;
   #Orz.Cin.Manager.Control_ON := #Vrt.Cin.Manager.Control_ON := #Cin.Manager.Control_ON;


   #Vrt.Cin.Manager.Rest := FALSE;
   #Vrt.Cin.Manager.Work := FALSE;
   #Orz.Cin.Manager.Rest := FALSE;
   #Orz.Cin.Manager.Work := FALSE;
   #Ax.CIn.Manager.MoveToPos := FALSE;


   // Operazione riposo del cilindro verticale ed orizzontale sullo spintore
   IF (#Ctrl.SpinVrtOrz.OP_Rest OR #Cin.Manager.REST_Req) AND #Sts.OP_Spin_Rest_Cnd THEN

       #Orz.Cin.Manager.Rest := #Orz.COut.Rest := TRUE;
       #Vrt.Cin.Manager.Rest := #Vrt.COut.Rest := #Orz.COut.Rest;

       // Operazione lavoro del cilindro verticale ed orizzontale sullo spintore   
   ELSIF (#Ctrl.SpinVrtOrz.OP_Work OR #Cin.Manager.WORK_Req) AND #Sts.OP_Spin_Work_Cnd THEN

       #Vrt.Cin.Manager.Work := #Vrt.COut.Work := TRUE;
       #Orz.Cin.Manager.Work := #Vrt.Cin.Manager.Work;

   END_IF;

   // Operazione arresto dell' asse spintore quando i 2 ciclindri sono in riposo
   IF #Ctrl.Ax.OP_Rest AND #Sts.OP_Ax_Rest_Cnd THEN
       #Ax.CIn.Manager.Pos := #Data.Ax_Pos.PosAttesa;
       #Ax.CIn.Manager.Vel := #Par_Ax_Auto.Aut_Vel;
       #Ax.CIn.Manager.Acc := #Par_Ax_Auto.Aut_Acc;
       #Ax.CIn.Manager.Dec := #Par_Ax_Auto.Aut_Dec;
       #Ax.CIn.Manager.MoveToPos := TRUE;

       // Se raggiungo la pos.attesa spengo il comando
   ELSIF #Ctrl.Ax.OP_Rest AND #Sts.OP_Ax_Rest_Cnd AND #COut.Ax_Sts.PosAttesa_Reached THEN
       #Ax.CIn.Manager.MoveToPos := #Ax.CIn.Manager.Control_ON := FALSE;

   END_IF;

   // Operazione lavoro dell' asse spintore quando i 2 ciclindri sono in lavoro
   IF #Ctrl.Ax.OP_Work AND #Sts.OP_Ax_Work_Cnd AND #Vrt.COut.Work AND #Orz.COut.Work
        AND NOT #Alarm.Orz_AnalSens_Compressed THEN
       #Ax.CIn.Manager.Pos := #Data.Ax_Pos.PosFineSpinta;
       #Ax.CIn.Manager.Vel := #Par_Ax_Auto.Aut_Vel;
       #Ax.CIn.Manager.Acc := #Par_Ax_Auto.Aut_Acc;
       #Ax.CIn.Manager.Dec := #Par_Ax_Auto.Aut_Dec;
       #Ax.CIn.Manager.MoveToPos := TRUE;

      // Se raggiungo la pos. o il sensore viene compresso disabilito la spinta 
   ELSIF (#Ctrl.Ax.OP_Work AND #Sts.OP_Ax_Work_Cnd) AND #COut.Ax_Sts.PosFineSpinta_Reached THEN
       #Ax.CIn.Manager.MoveToPos := FALSE;

   ELSIF (#Ctrl.Ax.OP_Work AND #Sts.OP_Ax_Work_Cnd) AND #Alarm.Orz_AnalSens_Compressed THEN
       #Ax.CIn.Manager.MoveToPos := FALSE;

   END_IF;
END_REGION

REGION Network 21 (SCL): Verticale + Orizzontale + Ax - CIn Abilitazioni Stop Manager
   #Vrt.Cin.Manager.EnableStopDoorOpeningReq := #Orz.Cin.Manager.EnableStopDoorOpeningReq
   := #Ax.CIn.Manager.EnableStopDoorOpeningReq := #Cin.Manager.EnableStopDoorOpeningReq;

   #Vrt.Cin.Manager.EnableStopInPhase := #Orz.Cin.Manager.EnableStopInPhase
   := #Ax.CIn.Manager.EnableStopInPhase := #Cin.Manager.EnableStopInPhase;

   #Vrt.Cin.Manager.EnableStopProgrammed := #Orz.Cin.Manager.EnableStopProgrammed
   := #Ax.CIn.Manager.EnableStopProgrammed := #Cin.Manager.EnableStopProgrammed;
END_REGION

REGION Network 22: <+>
END_REGION

REGION Network 23: Warning manacanza condizioni esecuzione Operazione RIPOSO / LAVORO
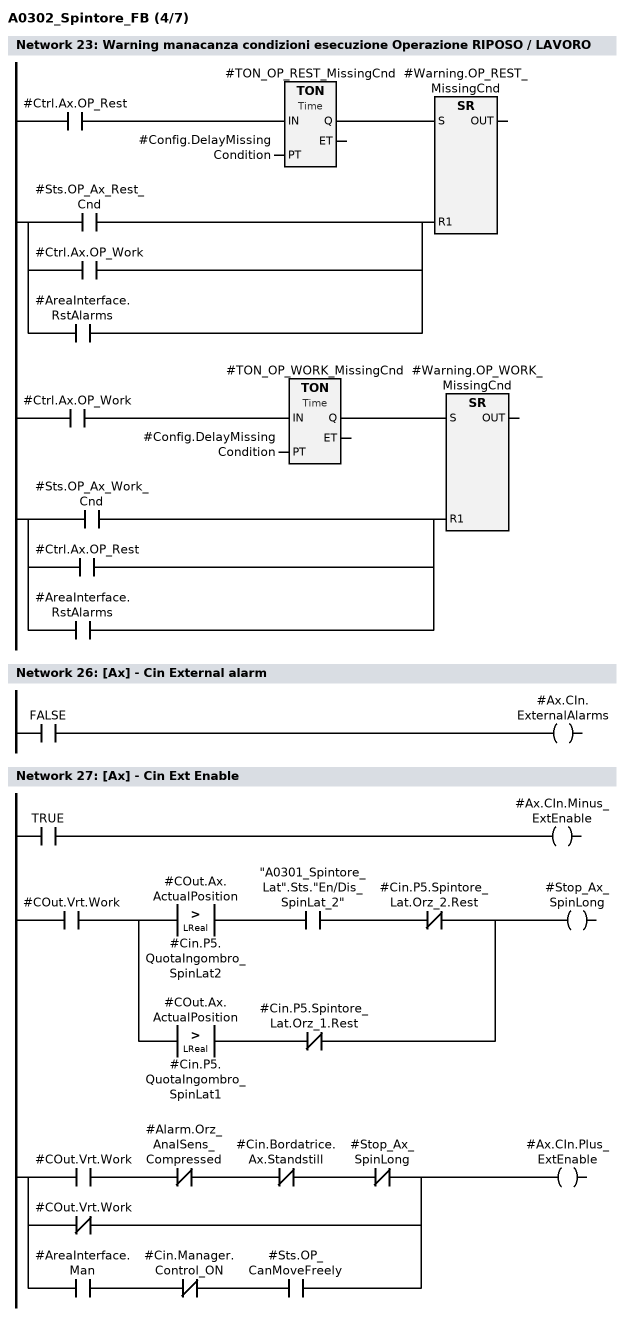
   RUNG wire#powerrail
      Contact( #Ctrl.Ax.OP_Rest )
      { S7_Templates := "time_type := Time" } #TON_OP_REST_MissingCnd.TON(pt := #Config.DelayMissingCondition, et =>)
      S_SR(operand := #Warning.OP_REST_MissingCnd, r1 := wire#w1)
   END_RUNG
   RUNG wire#powerrail
      Contact( #Sts.OP_Ax_Rest_Cnd )
   END_RUNG wire#w1
   RUNG wire#powerrail
      Contact( #Ctrl.Ax.OP_Work )
   END_RUNG wire#w1
   RUNG wire#powerrail
      Contact( #AreaInterface.RstAlarms )
   END_RUNG wire#w1
   RUNG wire#powerrail
      Contact( #Ctrl.Ax.OP_Work )
      { S7_Templates := "time_type := Time" } #TON_OP_WORK_MissingCnd.TON(pt := #Config.DelayMissingCondition, et =>)
      S_SR(operand := #Warning.OP_WORK_MissingCnd, r1 := wire#w2)
   END_RUNG
   RUNG wire#powerrail
      Contact( #Sts.OP_Ax_Work_Cnd )
   END_RUNG wire#w2
   RUNG wire#powerrail
      Contact( #Ctrl.Ax.OP_Rest )
   END_RUNG wire#w2
   RUNG wire#powerrail
      Contact( #AreaInterface.RstAlarms )
   END_RUNG wire#w2
   // the same network as SCL:
   #TON_OP_REST_MissingCnd(IN := #Ctrl.Ax.OP_Rest, PT := #Config.DelayMissingCondition);   // TON
   IF #TON_OP_REST_MissingCnd.Q THEN
       #Warning.OP_REST_MissingCnd := TRUE;   // SR flip-flop
   END_IF;
   IF #Sts.OP_Ax_Rest_Cnd OR #Ctrl.Ax.OP_Work OR #AreaInterface.RstAlarms THEN
       #Warning.OP_REST_MissingCnd := FALSE;
   END_IF;
   #TON_OP_WORK_MissingCnd(IN := #Ctrl.Ax.OP_Work, PT := #Config.DelayMissingCondition);   // TON
   IF #TON_OP_WORK_MissingCnd.Q THEN
       #Warning.OP_WORK_MissingCnd := TRUE;   // SR flip-flop
   END_IF;
   IF #Sts.OP_Ax_Work_Cnd OR #Ctrl.Ax.OP_Rest OR #AreaInterface.RstAlarms THEN
       #Warning.OP_WORK_MissingCnd := FALSE;
   END_IF;
END_REGION

REGION Network 25 (SCL): << RIFERIMENTI [Spintore Ax] - Positioning Manager >>
   // ******************************************************************************************
   REGION // TRASFERIMENTO DELLE RAMPE

       // Rampe in Automatico o Semi-Automatico
       IF #AreaInterface.Aut AND NOT #Cin.SemiAut_Pb THEN
           #Ax.CIn.Manager.Acc := #Par_Ax_Auto.Aut_Acc;
           #Ax.CIn.Manager.Dec := #Par_Ax_Auto.Aut_Dec;
       ELSIF #Cin.SemiAut_Pb THEN
           #Ax.CIn.Manager.Acc := #Par_Ax_Auto.Aut_Acc;
           #Ax.CIn.Manager.Dec := #Par_Ax_Auto.Aut_Dec;
       END_IF;

       // Rampe in Manuale
       IF #AreaInterface.Man AND NOT #Cin.SemiAut_Pb THEN
           #Ax.CIn.Manager.Acc := #Par_Ax_Manu.Man_Acc;
           #Ax.CIn.Manager.Dec := #Par_Ax_Manu.Man_Dec;
       END_IF;
   END_REGION

   // ******************************************************************************************
   REGION // // CALCOLO DELLA VELOCITA' TRASFERITA AL DRIVE IN BASE AL CALCOLO DEL CICLINDRO COMPENSATORE
       (*
   #Sts.ResiduoCilindro := #CorsaCilindro - #Sts.PosCilindro;

   #Sts.spazio_frenata := ((#Ctrl.Vel / 60.0) ** 2.0) /(2.0 * #Ctrl.Dec);

   #SpazioSafe := #Sts.spazio_frenata + #Par.CylComp_SafeResidual;

   #Ctrl.StopSicurezza := (#Sts.ResiduoCilindro - #SpazioSafe) < 0.0;

   // bisogna calcolare la decelerazione massima per rispettare frenata
   // 
   #Sts.DecMassima := ((#Ctrl.Vel / 60.0) ** 2.0) / (2 * (#Sts.ResiduoCilindro - #Par.CylComp_SafeResidual));
   *)

       // Velocità asse in base alla velocità della chiudi bordi..
       #Ctrl.Ax.Vel := #Cin.Bordatrice.TargetVel * #Cin.Bordatrice.Perc_Vel / 100.0;

       // Limite decellerazione dell'asse
       #DecMax := (#Ax.Config.Ax.MaxDec_S120_P2573 / 1000.0);

   (*// Spazio di frenata da raggiungere
   // 
   #SpazioSafe := #CorsaCilindroCompensatore - #Par.Spintore.Compensatore_SpazioResiduoExtra;
   *)

       // Nuovo valore di velocità per limitare e rispettare spazio di arresto con massima decelerazione possibile
       // 
       #Ctrl.Ax.VelMax := LREAL_TO_REAL(IN:= (60.0 * (SQRT(2.0 * #DecMax * #Orz_SpazioSafe))));

       // Limitazione della velocità per rispettare lo spazio di frenata   
       #Ctrl.Ax.Vel := MIN_REAL(IN1 := #Ctrl.Ax.Vel, IN2 := #Ctrl.Ax.VelMax);

   END_REGION ;

   // *****************************************************************************************
   REGION // CALCOLO DELLA VELOCITA' E TRASFERIMENTO IN BASE ALLO STATO IMPIANTO
       //
       IF NOT #Ax.CIn.Manager.Control_ON THEN
           // CALCOLO VELOCITA' IN BASE ALL'OVERIDE
           IF #Ax.AreaInterface.Aut THEN
               #Ax.CIn.Manager.Vel := #Ctrl.Ax.Vel;
           ELSIF #Cin.SemiAut_Pb THEN
               #Ax.CIn.Manager.Vel := (#Par_Ax_Auto.SemiAut_Vel * #Ctrl.Ax.Vel);
           END_IF;
       END_IF;
   END_REGION ;
END_REGION

REGION Network 26: [Ax] - Cin External alarm
   RUNG wire#powerrail
      Contact( FALSE )
      Coil( #Ax.CIn.ExternalAlarms )
   END_RUNG
   // the same network as SCL:
   #Ax.CIn.ExternalAlarms := FALSE;
END_REGION

REGION Network 27: [Ax] - Cin Ext Enable
   RUNG wire#powerrail
      Contact( TRUE )
      Coil( #Ax.CIn.Minus_ExtEnable )
   END_RUNG
   RUNG wire#powerrail
      Contact( #COut.Vrt.Work )
      wire#w1
      { S7_Templates := "SrcType := LReal" } GT_Contact(in1 := #COut.Ax.ActualPosition, in2 := #Cin.P5.QuotaIngombro_SpinLat2)
      Contact( "A0301_Spintore_Lat".Sts."En/Dis_SpinLat_2" )
      I_Contact( #Cin.P5.Spintore_Lat.Orz_2.Rest )
      wire#w2
      Coil( #Stop_Ax_SpinLong )
   END_RUNG
   RUNG wire#w1
      { S7_Templates := "SrcType := LReal" } GT_Contact(in1 := #COut.Ax.ActualPosition, in2 := #Cin.P5.QuotaIngombro_SpinLat1)
      I_Contact( #Cin.P5.Spintore_Lat.Orz_1.Rest )
   END_RUNG wire#w2
   RUNG wire#powerrail
      Contact( #COut.Vrt.Work )
      I_Contact( #Alarm.Orz_AnalSens_Compressed )
      I_Contact( #Cin.Bordatrice.Ax.Standstill )
      I_Contact( #Stop_Ax_SpinLong )
      wire#w3
      Coil( #Ax.CIn.Plus_ExtEnable )
   END_RUNG
   RUNG wire#powerrail
      I_Contact( #COut.Vrt.Work )
   END_RUNG wire#w3
   RUNG wire#powerrail
      Contact( #AreaInterface.Man )
      I_Contact( #Cin.Manager.Control_ON )
      Contact( #Sts.OP_CanMoveFreely )
   END_RUNG wire#w3
   // the same network as SCL:
   #Ax.CIn.Minus_ExtEnable := TRUE;
   #Stop_Ax_SpinLong := #COut.Vrt.Work AND (((#COut.Ax.ActualPosition > #Cin.P5.QuotaIngombro_SpinLat2) AND "A0301_Spintore_Lat".Sts."En/Dis_SpinLat_2" AND NOT #Cin.P5.Spintore_Lat.Orz_2.Rest) OR ((#COut.Ax.ActualPosition > #Cin.P5.QuotaIngombro_SpinLat1) AND NOT #Cin.P5.Spintore_Lat.Orz_1.Rest));
   #Ax.CIn.Plus_ExtEnable := (#COut.Vrt.Work AND NOT #Alarm.Orz_AnalSens_Compressed AND NOT #Cin.Bordatrice.Ax.Standstill AND NOT #Stop_Ax_SpinLong) OR NOT #COut.Vrt.Work OR (#AreaInterface.Man AND NOT #Cin.Manager.Control_ON AND #Sts.OP_CanMoveFreely);
END_REGION

REGION Network 28: [Ax] HMI preset position
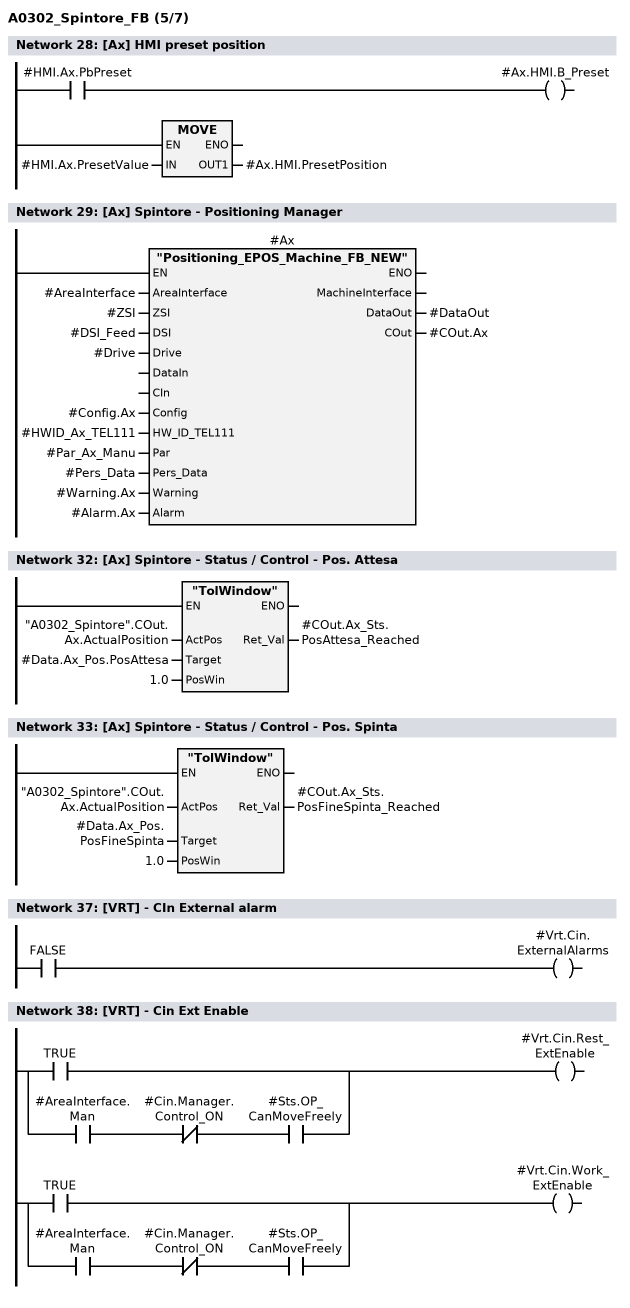
   RUNG wire#powerrail
      Contact( #HMI.Ax.PbPreset )
      Coil( #Ax.HMI.B_Preset )
   END_RUNG
   RUNG wire#powerrail
      Move(in := #HMI.Ax.PresetValue, out1 => #Ax.HMI.PresetPosition)
   END_RUNG
   // the same network as SCL:
   #Ax.HMI.B_Preset := #HMI.Ax.PbPreset;
   #Ax.HMI.PresetPosition := #HMI.Ax.PresetValue;
END_REGION

REGION Network 29: [Ax] Spintore - Positioning Manager
   RUNG wire#powerrail
      #Ax(AreaInterface := #AreaInterface, ZSI := #ZSI, DSI := #DSI_Feed, Drive := #Drive, DataIn :=, CIn :=, Config := #Config.Ax, HW_ID_TEL111 := #HWID_Ax_TEL111, Par := #Par_Ax_Manu, Pers_Data := #Pers_Data, Warning := #Warning.Ax, Alarm := #Alarm.Ax, MachineInterface =>, DataOut => #DataOut, COut => #COut.Ax)
   END_RUNG
   // the same network as SCL:
   #Ax(AreaInterface := #AreaInterface,   // "Positioning_EPOS_Machine_FB_NEW"
       ZSI := #ZSI,
       DSI := #DSI_Feed,
       Drive := #Drive,
       Config := #Config.Ax,
       HW_ID_TEL111 := #HWID_Ax_TEL111,
       Par := #Par_Ax_Manu,
       Pers_Data := #Pers_Data,
       Warning := #Warning.Ax,
       Alarm := #Alarm.Ax,
       DataOut => #DataOut,
       COut => #COut.Ax);
END_REGION

REGION Network 30: <+>
END_REGION

REGION Network 31: <<< CONTROLLO REQ da TRAKING E CAMBIO POS. >>>
END_REGION

REGION Network 32: [Ax] Spintore - Status / Control - Pos. Attesa
   RUNG wire#powerrail
      "TolWindow"(ActPos := "A0302_Spintore".COut.Ax.ActualPosition, Target := #Data.Ax_Pos.PosAttesa, PosWin := 1.0, Ret_Val => #COut.Ax_Sts.PosAttesa_Reached)
   END_RUNG
   // the same network as SCL:
   #COut.Ax_Sts.PosAttesa_Reached := "TolWindow"(ActPos := "A0302_Spintore".COut.Ax.ActualPosition,
                           Target := #Data.Ax_Pos.PosAttesa,
                           PosWin := 1.0);
END_REGION

REGION Network 33: [Ax] Spintore - Status / Control - Pos. Spinta
   RUNG wire#powerrail
      "TolWindow"(ActPos := "A0302_Spintore".COut.Ax.ActualPosition, Target := #Data.Ax_Pos.PosFineSpinta, PosWin := 1.0, Ret_Val => #COut.Ax_Sts.PosFineSpinta_Reached)
   END_RUNG
   // the same network as SCL:
   #COut.Ax_Sts.PosFineSpinta_Reached := "TolWindow"(ActPos := "A0302_Spintore".COut.Ax.ActualPosition,
                           Target := #Data.Ax_Pos.PosFineSpinta,
                           PosWin := 1.0);
END_REGION

REGION Network 34: <+>
END_REGION

REGION Network 36: <<< SPINTORE LONGITUDINALE - VRT >>>
END_REGION

REGION Network 37: [VRT] - CIn External alarm
   RUNG wire#powerrail
      Contact( FALSE )
      Coil( #Vrt.Cin.ExternalAlarms )
   END_RUNG
   // the same network as SCL:
   #Vrt.Cin.ExternalAlarms := FALSE;
END_REGION

REGION Network 38: [VRT] - Cin Ext Enable
   RUNG wire#powerrail
      Contact( TRUE )
      wire#w1
      Coil( #Vrt.Cin.Rest_ExtEnable )
   END_RUNG
   RUNG wire#powerrail
      Contact( #AreaInterface.Man )
      I_Contact( #Cin.Manager.Control_ON )
      Contact( #Sts.OP_CanMoveFreely )
   END_RUNG wire#w1
   RUNG wire#powerrail
      Contact( TRUE )
      wire#w2
      Coil( #Vrt.Cin.Work_ExtEnable )
   END_RUNG
   RUNG wire#powerrail
      Contact( #AreaInterface.Man )
      I_Contact( #Cin.Manager.Control_ON )
      Contact( #Sts.OP_CanMoveFreely )
   END_RUNG wire#w2
   // the same network as SCL:
   #Vrt.Cin.Rest_ExtEnable := TRUE OR (#AreaInterface.Man AND NOT #Cin.Manager.Control_ON AND #Sts.OP_CanMoveFreely);
   #Vrt.Cin.Work_ExtEnable := TRUE OR (#AreaInterface.Man AND NOT #Cin.Manager.Control_ON AND #Sts.OP_CanMoveFreely);
END_REGION

REGION Network 39: [VRT] - Valve Manager
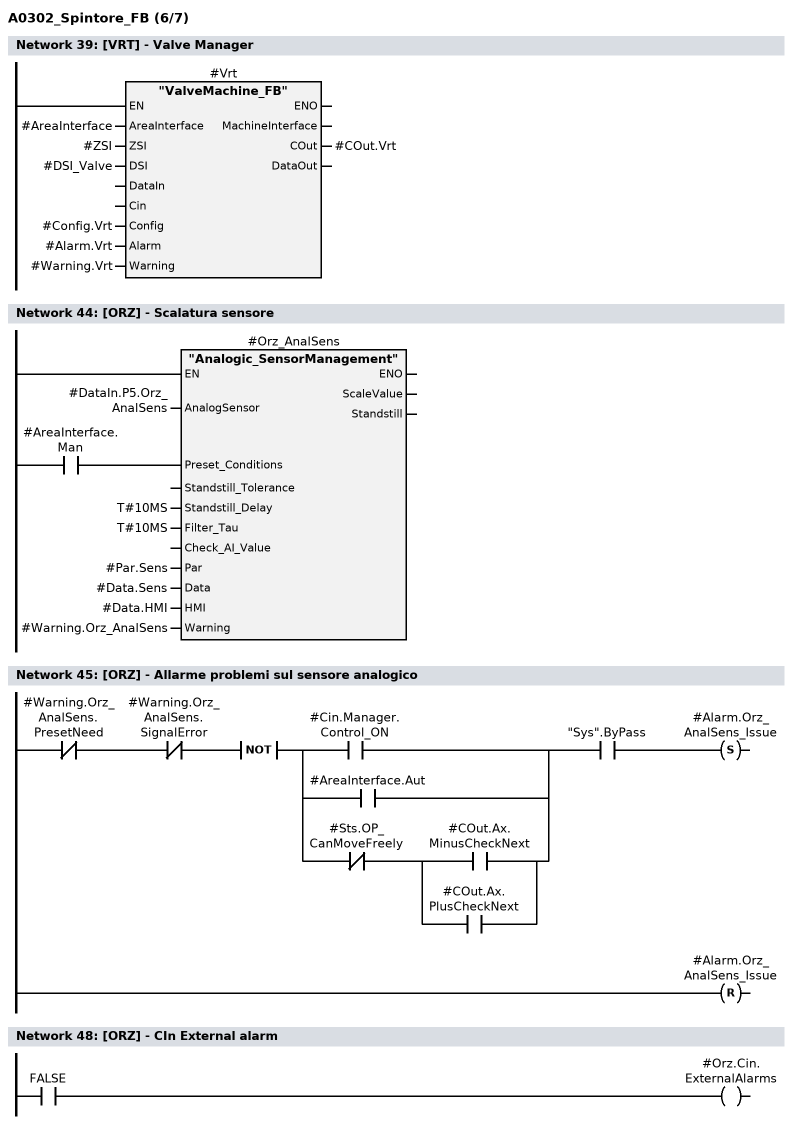
   RUNG wire#powerrail
      #Vrt(AreaInterface := #AreaInterface, ZSI := #ZSI, DSI := #DSI_Valve, DataIn :=, Cin :=, Config := #Config.Vrt, Alarm := #Alarm.Vrt, Warning := #Warning.Vrt, MachineInterface =>, COut => #COut.Vrt, DataOut =>)
   END_RUNG
   // the same network as SCL:
   #Vrt(AreaInterface := #AreaInterface,   // "ValveMachine_FB"
        ZSI := #ZSI,
        DSI := #DSI_Valve,
        Config := #Config.Vrt,
        Alarm := #Alarm.Vrt,
        Warning := #Warning.Vrt,
        COut => #COut.Vrt);
END_REGION

REGION Network 41: <<< SPINTORE LONGITUDINALE - ORZ >>>
END_REGION

REGION Network 42: <+>
END_REGION

REGION Network 43: << GESTIONE SPINTORE ORIZ ANALOGIC SENSOR >>
END_REGION

REGION Network 44: [ORZ] - Scalatura sensore
   RUNG wire#powerrail
      #Orz_AnalSens(Preset_Conditions := wire#w1, AnalogSensor := #DataIn.P5.Orz_AnalSens, Standstill_Tolerance :=, Standstill_Delay := T#10MS, Filter_Tau := T#10MS, Check_AI_Value :=, Par := #Par.Sens, Data := #Data.Sens, HMI := #Data.HMI, Warning := #Warning.Orz_AnalSens, ScaleValue =>, Standstill =>)
   END_RUNG
   RUNG wire#powerrail
      Contact( #AreaInterface.Man )
   END_RUNG wire#w1
   // the same network as SCL:
   #Orz_AnalSens(AnalogSensor := #DataIn.P5.Orz_AnalSens,   // "Analogic_SensorManagement"
                 Preset_Conditions := #AreaInterface.Man,
                 Standstill_Delay := T#10MS,
                 Filter_Tau := T#10MS,
                 Par := #Par.Sens,
                 Data := #Data.Sens,
                 HMI := #Data.HMI,
                 Warning := #Warning.Orz_AnalSens);
END_REGION

REGION Network 45: [ORZ] - Allarme problemi sul sensore analogico
   RUNG wire#powerrail
      I_Contact( #Warning.Orz_AnalSens.PresetNeed )
      I_Contact( #Warning.Orz_AnalSens.SignalError )
      Not()
      wire#w1
      Contact( #Cin.Manager.Control_ON )
      wire#w2
      Contact( "Sys".ByPass )
      S_Coil( #Alarm.Orz_AnalSens_Issue )
   END_RUNG
   RUNG wire#w1
      Contact( #AreaInterface.Aut )
   END_RUNG wire#w2
   RUNG wire#w1
      I_Contact( #Sts.OP_CanMoveFreely )
      wire#w3
      Contact( #COut.Ax.MinusCheckNext )
   END_RUNG wire#w2
   RUNG wire#w3
      Contact( #COut.Ax.PlusCheckNext )
   END_RUNG wire#w2
   RUNG wire#powerrail
      R_Coil( #Alarm.Orz_AnalSens_Issue )
   END_RUNG
   // the same network as SCL:
   IF NOT (NOT #Warning.Orz_AnalSens.PresetNeed AND NOT #Warning.Orz_AnalSens.SignalError) AND (#Cin.Manager.Control_ON OR #AreaInterface.Aut OR (NOT #Sts.OP_CanMoveFreely AND (#COut.Ax.MinusCheckNext OR #COut.Ax.PlusCheckNext))) AND "Sys".ByPass THEN
       #Alarm.Orz_AnalSens_Issue := TRUE;
   END_IF;
   #Alarm.Orz_AnalSens_Issue := FALSE;
END_REGION

REGION Network 46 (SCL): [ORZ] - Calcolo range lavoro sensore
       // ********************************************************************************************************************************************
       // Calcolo lo spazio di sicurezza se ho eseguito il preset del sensore
       // Spazio di frenata da raggiungere

       IF #Par.Sens.Enable THEN
           IF #Data.Sens.OffsetValid THEN
               #Orz_SpazioSafe := #Par.Sens.RangeHigh - #Par_Mach.Tol_Work  ;
           END_IF;

           // Controllo finestra di lavoro del sensore, dato il valore di lavoro sicuro,se è inferiore sino in compressione sul pezzo.  
           IF  #Data.Sens.OffsetValid AND #Orz_SpazioSafe <> 0 AND 
               (#Orz_AnalSens.ScaleValue < (#Par.Sens.RangeHigh - #Orz_SpazioSafe)) THEN
               #Alarm.Orz_AnalSens_Compressed := 1;
           ELSE
               #Alarm.Orz_AnalSens_Compressed := 0;
           END_IF;
       END_IF;
END_REGION

REGION Network 47: <+>
END_REGION

REGION Network 48: [ORZ] - CIn External alarm
   RUNG wire#powerrail
      Contact( FALSE )
      Coil( #Orz.Cin.ExternalAlarms )
   END_RUNG
   // the same network as SCL:
   #Orz.Cin.ExternalAlarms := FALSE;
END_REGION

REGION Network 49: [ORZ] - Cin Ext Enable
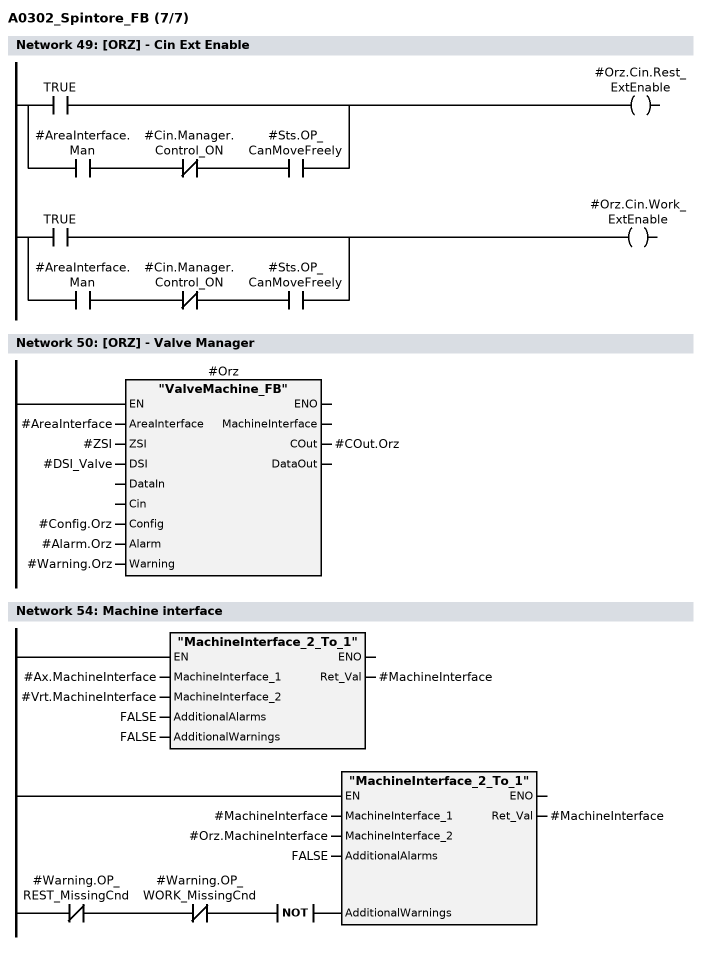
   RUNG wire#powerrail
      Contact( TRUE )
      wire#w1
      Coil( #Orz.Cin.Rest_ExtEnable )
   END_RUNG
   RUNG wire#powerrail
      Contact( #AreaInterface.Man )
      I_Contact( #Cin.Manager.Control_ON )
      Contact( #Sts.OP_CanMoveFreely )
   END_RUNG wire#w1
   RUNG wire#powerrail
      Contact( TRUE )
      wire#w2
      Coil( #Orz.Cin.Work_ExtEnable )
   END_RUNG
   RUNG wire#powerrail
      Contact( #AreaInterface.Man )
      I_Contact( #Cin.Manager.Control_ON )
      Contact( #Sts.OP_CanMoveFreely )
   END_RUNG wire#w2
   // the same network as SCL:
   #Orz.Cin.Rest_ExtEnable := TRUE OR (#AreaInterface.Man AND NOT #Cin.Manager.Control_ON AND #Sts.OP_CanMoveFreely);
   #Orz.Cin.Work_ExtEnable := TRUE OR (#AreaInterface.Man AND NOT #Cin.Manager.Control_ON AND #Sts.OP_CanMoveFreely);
END_REGION

REGION Network 50: [ORZ] - Valve Manager
   RUNG wire#powerrail
      #Orz(AreaInterface := #AreaInterface, ZSI := #ZSI, DSI := #DSI_Valve, DataIn :=, Cin :=, Config := #Config.Orz, Alarm := #Alarm.Orz, Warning := #Warning.Orz, MachineInterface =>, COut => #COut.Orz, DataOut =>)
   END_RUNG
   // the same network as SCL:
   #Orz(AreaInterface := #AreaInterface,   // "ValveMachine_FB"
        ZSI := #ZSI,
        DSI := #DSI_Valve,
        Config := #Config.Orz,
        Alarm := #Alarm.Orz,
        Warning := #Warning.Orz,
        COut => #COut.Orz);
END_REGION

REGION Network 51: <+>
END_REGION

REGION Network 52 (SCL): Stazione COut
   // VALVOLE SPINTORE
   #COut.Spintore.Standstill := #Vrt.COut.Standstill AND #Orz.COut.Standstill;
   #COut.Spintore.Rest_CheckNext := #Ctrl.Ax.OP_Rest AND #Ctrl.SpinVrtOrz.OP_Rest;
   #COut.Spintore.Work_CheckNext := #Ctrl.Ax.OP_Work AND #Ctrl.SpinVrtOrz.OP_Work ;
   #COut.Spintore.Rest := #Vrt.COut.Rest AND #Orz.COut.Rest;
   #COut.Spintore.Work := #Vrt.COut.Work AND #Orz.COut.Work;

   // SPINTORE LONGITUDINALE
   #COut.Ax := #Ax.COut;
   #COut.Vrt := #Vrt.COut;
   #COut.Orz := #Orz.COut;
END_REGION

REGION Network 53: <<< MACHINE STATUS >>>
END_REGION

REGION Network 54: Machine interface
   RUNG wire#powerrail
      "MachineInterface_2_To_1"(MachineInterface_1 := #Ax.MachineInterface, MachineInterface_2 := #Vrt.MachineInterface, AdditionalAlarms := FALSE, AdditionalWarnings := FALSE, Ret_Val => #MachineInterface)
   END_RUNG
   RUNG wire#powerrail
      "MachineInterface_2_To_1"(AdditionalWarnings := wire#w1, MachineInterface_1 := #MachineInterface, MachineInterface_2 := #Orz.MachineInterface, AdditionalAlarms := FALSE, Ret_Val => #MachineInterface)
   END_RUNG
   RUNG wire#powerrail
      I_Contact( #Warning.OP_REST_MissingCnd )
      I_Contact( #Warning.OP_WORK_MissingCnd )
      Not()
   END_RUNG wire#w1
   // the same network as SCL:
   #MachineInterface := "MachineInterface_2_To_1"(MachineInterface_1 := #Ax.MachineInterface,
                           MachineInterface_2 := #Vrt.MachineInterface,
                           AdditionalAlarms := FALSE,
                           AdditionalWarnings := FALSE);
   #MachineInterface := "MachineInterface_2_To_1"(MachineInterface_1 := #MachineInterface,
                           MachineInterface_2 := #Orz.MachineInterface,
                           AdditionalAlarms := FALSE,
                           AdditionalWarnings := NOT (NOT #Warning.OP_REST_MissingCnd AND NOT #Warning.OP_WORK_MissingCnd));
END_REGION
END_FUNCTION_BLOCK
